FUNCTION_BLOCK FB_ECS_Linear_AO
VAR_INPUT PERSISTENT
	bEnable									: BOOL;											//{#lynus.ag#()} //Enable the Fuctionblock and his logic
	bPowerDataInvers						: BOOL;											//With True its possible to invert all received power data from the electric meter
	bNoLinear								: BOOL;											//Output Power from the device is not linear. Use the Values from the Table Of Interpolation Points.
	byElectricFuseLine						: BYTE; 										//Electric Fuse Line on wich the ECS is connected => 1 2 3 (If 0 then this charging station is not connected to a Electric Fuse Line)
	diNrOfEMS_IN							: DINT;											//Number of EMS what control this Device.
	diNrOfEM_IN_CS							: DINT;											//Number of the electric meter for incoming power data. (Power Data for this Device)
	stSetupECS								: ST_Setup_ECS;									//{#lynus.ag#()} //Setup charging station
	arrTableOfInterpolationPoints			: ARRAY[1..10] OF REAL;							//Table Of Interpolation Points. Corresponds to the different power values in the non-linear curve of the device. The last value must correspond to the maximum power.
END_VAR
VAR_INPUT
	bCarConnectedExt						: BOOL;											//Car connected signal from external function			
	bErrorExt								: BOOL;											//Error Signal from external Function
	bWarningExt								: BOOL;											//Warning Signal from external Function 						
END_VAR
VAR_OUTPUT
	stDataECS								: ST_ECS_Output;								//{#lynus.ag#()} //Electric charging station output data
	diNrOfECS_OUT							: DINT;											//Active Number from the Electric charging Function for using on other functions
	rTargetPowerForExtFunc					: REAL;											//Target Power from 0% to +100% to use on a external Function
	rTargetChargCurrentForExtFunc			: REAL;											//Target charge Current to use on a external Function
END_VAR
VAR
	{attribute 'hide'}
	fbCS									: FB_ElectricChargingStation;					//Function block for electric charging station
	{attribute 'hide'}
	fbNumberDevice							: FB_NumberOfDevice;							//Function block to calcualte the number of the Device
	{attribute 'hide'}
	fbInterpolation							: FB_Lin_Interpolation;							//Function for interpolation
	fbDIExternalLock						: FB_XL1XXX_DI;									//Digital Input from external loock signal
	fbAOCS									: FB_XL4XXX_AO;									//Analog Output to swtich on and off the charging station
	{attribute 'hide'}
	timDissableFunctions					: TON;											//Timer to dissable the Function after Lynus_Standards.Constants_General.tTimeDissableLynusFunctions Days without connection to the Lynus Cloud
	{attribute 'hide'}
	timResetConnectionOnGVL					: TON;											//Timer to try reset the connection Flag on the GVL. (When somebody delete the Connection Function and make only a onlinechange)
	{attribute 'hide'}
	arrPD									: ARRAY[1..25] OF FB_PersistentData_Number;		//Function to save persistent data 
	{attribute 'hide'}
	byWaitInStep							: BYTE;											//Wait in Step before start to clean data on PLC
	{attribute 'hide'}
	iStateGVLData							: INT;											//State machine to handle the data on the GVL
	{attribute 'hide'}
	diNumberOfActiveBatterys				: DINT;											//Number of active batterys
	{attribute 'hide'}
	diNumberOfBatteryInverterInEPO			: DINT;											//Number of battery inverters that work in Emergency Power operation 
	{attribute 'hide'}
	diCounterForGVL							: DINT;											//Counter to clean old data on GVL
	{attribute 'hide'}
	diLPForGVL								: DINT;											//Loop to clean old data on GVL
	{attribute 'hide'}
	dwSumSOC								: DWORD;										//Sum of the SOC from all batterys	
	{attribute 'hide'}
	liLPBatteryData							: LINT;											//Loop to check some data from batterys
	{attribute 'hide'}
	liLPInEPO								: LINT;											//Loop to check if 1 or more battery inverters build a island grid
END_VAR
VAR PERSISTENT
	{attribute 'conditionalshow'}
	diNrOfEMS_IN_CP							: DINT;											//Number of EMS what control this Device to compare with the original
END_VAR

//Creator : Kai Ebensperger
//Company : Lynus AG
//Date : 19.05.2021
//Version : 1.0.0.0

//With this function block its possible to switch on and off a charging station
//Its also possible to control the target power with the analog output signal
//With the Nr from the Electric Meter its possible to send the data fromt the electric meter directly to the CS function to display it

//NOTE for diNr.....Designation => 
//_IN = Here Data come in from other Functions or go out to other functions about the GVL
//_OUT = Here Data go out to other functions about the GVL

(*------------------------------------------------------------Limits----------------------------------------------------------------------------------*)

diNrOfEMS_IN := LIMIT(0,diNrOfEMS_IN,Constants_Energy.diMaxNumberOfEMS);
	diNrOfEM_IN_CS := LIMIT(0,diNrOfEM_IN_CS,Constants_Energy.diMaxNumberOfElectricMeters);	
		byElectricFuseLine := LIMIT(0,byElectricFuseLine,30);	
			
(*------------------------------------------------------------------Power Data----------------------------------------------------------------------------*)

//Energy Session Input data
fbCS.bCalculateEnergySession := FALSE;
fbCS.arrSocketPowerECS[1] := 0;
fbCS.arrSocketPowerECS[2] := 0;
fbCS.arrSocketPowerECS[3] := 0;
fbCS.arrSocketPowerECS[4] := 0;
fbCS.arrSocketEnergySession[1] := 0;
fbCS.arrSocketEnergySession[2] := 0;
fbCS.arrSocketEnergySession[3] := 0;
fbCS.arrSocketEnergySession[4] := 0;

IF NOT bPowerDataInvers THEN
	fbCS.lrCounterEnergyT1_Consumption := Lynus_Standards.GVL_Energy.stDataElectricMeters[diNrOfEM_IN_CS].lrCounterEnergyT1_Production * 1000;
	fbCS.lrCounterEnergyT2_Consumption := Lynus_Standards.GVL_Energy.stDataElectricMeters[diNrOfEM_IN_CS].lrCounterEnergyT2_Production * 1000;
	fbCS.lrCounterEnergyT1_Production := Lynus_Standards.GVL_Energy.stDataElectricMeters[diNrOfEM_IN_CS].lrCounterEnergyT1_Consumption * 1000;
	fbCS.lrCounterEnergyT2_Production := Lynus_Standards.GVL_Energy.stDataElectricMeters[diNrOfEM_IN_CS].lrCounterEnergyT1_Consumption * 1000;
	fbCS.lrTotalCounterEnergy_Consumption := Lynus_Standards.GVL_Energy.stDataElectricMeters[diNrOfEM_IN_CS].lrTotalCounterEnergy_Production * 1000;
	fbCS.lrTotalCounterEnergy_Production := Lynus_Standards.GVL_Energy.stDataElectricMeters[diNrOfEM_IN_CS].lrTotalCounterEnergy_Consumption * 1000;
		fbCS.lrTotalPowerECS := (Lynus_Standards.GVL_Energy.stDataElectricMeters[diNrOfEM_IN_CS].lrPower * 1000) * - 1;
ELSE
	fbCS.lrCounterEnergyT1_Consumption := Lynus_Standards.GVL_Energy.stDataElectricMeters[diNrOfEM_IN_CS].lrCounterEnergyT1_Consumption * 1000;
	fbCS.lrCounterEnergyT2_Consumption := Lynus_Standards.GVL_Energy.stDataElectricMeters[diNrOfEM_IN_CS].lrCounterEnergyT2_Consumption * 1000;
	fbCS.lrCounterEnergyT1_Production := Lynus_Standards.GVL_Energy.stDataElectricMeters[diNrOfEM_IN_CS].lrCounterEnergyT1_Production * 1000;
	fbCS.lrCounterEnergyT2_Production := Lynus_Standards.GVL_Energy.stDataElectricMeters[diNrOfEM_IN_CS].lrCounterEnergyT2_Production * 1000;
	fbCS.lrTotalCounterEnergy_Consumption := Lynus_Standards.GVL_Energy.stDataElectricMeters[diNrOfEM_IN_CS].lrTotalCounterEnergy_Consumption * 1000;
	fbCS.lrTotalCounterEnergy_Production := Lynus_Standards.GVL_Energy.stDataElectricMeters[diNrOfEM_IN_CS].lrTotalCounterEnergy_Production * 1000;
		fbCS.lrTotalPowerECS := Lynus_Standards.GVL_Energy.stDataElectricMeters[diNrOfEM_IN_CS].lrPower * 1000;
END_IF

(*-------------------------------------------------------------Calcualte the number of ECS---------------------------------------------------------------*)

fbNumberDevice(
	diActualNumberOfDevices:= Lynus_Standards.GVL_Energy.stNumberOfDevices.diNumberOfECS, 
	diMaxNumberOfDevices:= Constants_Energy.diMaxNumberOfElectricChargingStations, 
	udiCounterOnlineChange:= TwinCAT_SystemInfoVarList._AppInfo.OnlineChangeCnt, 
	bNumberIsCalculatet=> , 
	bFPNumberIsCalculatet=> , 
	bOnlineChange=> , 
	diNumberForThisDevice=> diNrOfECS_OUT, 
	diNumberOfTotalDevices=> );

//Write new Numer on GVL
IF fbNumberDevice.bFPNumberIsCalculatet THEN
	Lynus_Standards.GVL_Energy.stNumberOfDevices.diNumberOfECS := fbNumberDevice.diNumberOfTotalDevices;	
END_IF 

//Delete old Number on GVL
IF fbNumberDevice.bOnlineChange THEN 
	Lynus_Standards.GVL_Energy.stNumberOfDevices.diNumberOfECS := diNrOfECS_OUT;	
		iStateGVLData := 1; 
END_IF

(*-------------------------------------------------------------Service from Backend is ready and check the connection to backend for dissabel/enable Function---------------------------------------------------------------*)

//Try to reset the variable for connection on the GVL. When all is normal then the Lynus Mqtt connection function set this variable to true in the next cycle
//When we have no connection to the backend then after Lynus_Standards.Constants_General.tTimeDissableLynusFunctions days the Function is dissabled with all of his functionalities
timResetConnectionOnGVL(IN:= NOT timResetConnectionOnGVL.Q, PT:= T#1H, Q=> , ET=> );
	IF timResetConnectionOnGVL.Q THEN Lynus_Standards.GVL_Communicator.bStateConnectionToEnableFunctions := FALSE; END_IF
		IF NOT Lynus_Standards.GVL_Communicator.bStateConnectionToEnableFunctions THEN timDissableFunctions.IN := TRUE; ELSE timDissableFunctions.IN := FALSE; END_IF  
			timDissableFunctions(IN:= , PT:= Lynus_Standards.Constants_General.tTimeDissableLynusFunctions, Q=> , ET=> );	

(*------------------------------------------------------------------Error and Warning----------------------------------------------------------------------------*)	

IF timDissableFunctions.Q OR bWarningExt THEN fbCS.bWarning := TRUE; ELSE fbCS.bWarning := FALSE; END_IF   
	IF Lynus_Standards.GVL_Energy.stNumberOfDevices.diNumberOfECS > Constants_Energy.diMaxNumberOfElectricChargingStations OR bErrorExt THEN 
		fbCS.bError := TRUE;
	ELSE 
		fbCS.bError := FALSE;
	END_IF

IF timDissableFunctions.Q THEN fbCS.iWarningCode := 0;
ELSIF bWarningExt THEN fbCS.iWarningCode := 1;
END_IF

IF Lynus_Standards.GVL_Energy.stNumberOfDevices.diNumberOfECS > Constants_Energy.diMaxNumberOfElectricChargingStations THEN fbCS.iErrorCode := 1;
ELSIF bErrorExt THEN fbCS.iErrorCode := 0;
END_IF        	
	
(*------------------------------------------------------------------Logic----------------------------------------------------------------------------*)

//Calcualte the total SOC if we have more then 1 battery in our system
diNumberOfActiveBatterys := 0;
	dwSumSOC := 0;
		FOR liLPBatteryData := 1 TO Constants_Energy.diMaxNumberOfBatterys BY 1 DO
			IF Lynus_Standards.GVL_Energy.stDataOfBatterys[diNrOfEMS_IN,liLPBatteryData].bEnabled THEN diNumberOfActiveBatterys := diNumberOfActiveBatterys + 1; END_IF
				dwSumSOC := dwSumSOC + Lynus_Standards.GVL_Energy.stDataOfBatterys[diNrOfEMS_IN,liLPBatteryData].dwSOC;
		END_FOR
	
IF diNumberOfActiveBatterys > 0 THEN
	fbCS.dwBatterySOC := DINT_TO_DWORD(DWORD_TO_DINT(dwSumSOC) / diNumberOfActiveBatterys);
ELSE
	fbCS.dwBatterySOC := 100;	//When we have no battery in the ems system
END_IF

//Check if one or more Batterysystems or batteryinverter make island mode
diNumberOfBatteryInverterInEPO := 0;
	FOR liLPInEPO := 1 TO Constants_Energy.diMaxNumberOfBatteryInverters BY 1 DO
		IF Lynus_Standards.GVL_Energy.stDataOfBatteryInverters[diNrOfEMS_IN,liLPInEPO].bWorkOnIslandMode THEN fbCS.bEPOIsActive := TRUE; diNumberOfBatteryInverterInEPO := diNumberOfBatteryInverterInEPO + 1; END_IF
	END_FOR 
		IF diNumberOfBatteryInverterInEPO <= 0 THEN fbCS.bEPOIsActive := FALSE; END_IF

//Digital input for external lock signal
fbDIExternalLock(bInvers:= FALSE, bSignal=> );

//Car SOC, charging Time and Mode 3
fbCS.arrSOCCar[1] := 0;
fbCS.arrSOCCar[2] := 0;
fbCS.arrSOCCar[3] := 0;
fbCS.arrSOCCar[4] := 0;
	fbCS.arrSocketChargingTimeInput[1] := 0;
	fbCS.arrSocketChargingTimeInput[2] := 0;
	fbCS.arrSocketChargingTimeInput[3] := 0;
	fbCS.arrSocketChargingTimeInput[4] := 0;
		fbCS.arrSocketMode3StateECS[1] := '';
		fbCS.arrSocketMode3StateECS[2] := '';
		fbCS.arrSocketMode3StateECS[3] := '';
		fbCS.arrSocketMode3StateECS[4] := '';
	
//Functionblock ECS
fbCS(
	bEnable:= bEnable AND NOT timDissableFunctions.Q, 
	bError:= , 
	bEPOIsActive:= , 
	bExternalLock:= fbDIExternalLock.bSignal, 
	bCarConnected:= bCarConnectedExt, 
	bWriteWithDelay:= TRUE, 
	bCalculateEnergySession:= ,
	iErrorCode:= , 
	iWarningCode:= , 
	arrSocketChargingTimeInput:= , 
	arrSOCCar:= , 
	dwBatterySOC:= , 
	lrTotalCounterEnergy_Consumption:= , 
	lrTotalCounterEnergy_Production:= , 
	lrCounterEnergyT1_Consumption:= , 
	lrCounterEnergyT2_Consumption:= , 
	lrCounterEnergyT1_Production:= , 
	lrCounterEnergyT2_Production:= , 
	lrTotalPowerECS:= , 
	arrSocketEnergySession:= ,
	rTargetPower:= Lynus_Standards.GVL_Energy.stDataElectricChargingStations[diNrOfEMS_IN,diNrOfECS_OUT].rTargetPowerEMS, 
	rSupplyVoltage:= 692, 
	rMinCurrent:= 0, 
	tTimDelayOutput:= T#5S, 
	tDelayError:= T#5S,
	arrSocketMode3StateECS:= ,
	arrSocketPowerECS:= ,
	stSetupECS:= stSetupECS, 
	stDataECSOut=> , 
	stDataECSOutDelay=> stDataECS);	
	
(*-------------------------------------------------------------------------Output----------------------------------------------------------------------*)

IF bNoLinear THEN 
	fbInterpolation.rXInputValue := (stSetupECS.rMaxPower * fbCS.stDataECSOut.rTargetPower) / 100; 
		fbInterpolation.arrYIntermediateValues[1] := 10;
			fbInterpolation.arrYIntermediateValues[2] := 20;
				fbInterpolation.arrYIntermediateValues[3] := 30;
					fbInterpolation.arrYIntermediateValues[4] := 40;
						fbInterpolation.arrYIntermediateValues[5] := 50;
	fbInterpolation.arrYIntermediateValues[6] := 60;
		fbInterpolation.arrYIntermediateValues[7] := 70;
			fbInterpolation.arrYIntermediateValues[8] := 80;
				fbInterpolation.arrYIntermediateValues[9] := 90;
					fbInterpolation.arrYIntermediateValues[10] := 100;
	fbInterpolation(rXInputValue:=, arrXIntermediateValues:= arrTableOfInterpolationPoints, arrYIntermediateValues:=, rYOutputValue=> );
END_IF

IF bNoLinear THEN 
	fbAOCS.rSignal := fbInterpolation.rYOutputValue;
	//Target Power, to use this on a external Function
	rTargetPowerForExtFunc := fbInterpolation.rYOutputValue;
	rTargetChargCurrentForExtFunc := (fbCS.stDataECSOut.rTargetChargeCurrent * rTargetPowerForExtFunc) / 100; 
ELSE
	fbAOCS.rSignal := fbCS.stDataECSOut.rTargetPower;
	//Target Power, to use this on a external Function
	rTargetPowerForExtFunc := fbCS.stDataECSOut.rTargetPower;
	rTargetChargCurrentForExtFunc := fbCS.stDataECSOut.rTargetChargeCurrent;
END_IF

fbAOCS(
	rYMinTerminalValue:= 0, 
	rXMinInputSignal:= 0, 
	rYMaxTerminalValue:= 32767, 
	rXMaxInputSignal:= 100, 
	rSignal:= , 
	usiState=> );
							
(*-----------------------------------------------------------Handle data to Global structure for electric charging stations-----------------------------------------------------------------*)

//Delte al old Data on GVL after a online change or change on the variable diNrOfEMS_IDOD
IF diNrOfEMS_IN <> diNrOfEMS_IN_CP AND iStateGVLData = 0 THEN iStateGVLData := 10; END_IF 

CASE iStateGVLData OF
	
	0://Init Step
		byWaitInStep := 0;
			diCounterForGVL := 1;
	
	1://Wait for 4 Steps before clean al Data on GVL
		byWaitInStep := byWaitInStep + 1;
			IF byWaitInStep >= 4 AND fbNumberDevice.bNumberIsCalculatet THEN iStateGVLData := 2; END_IF
				//To much Devices, back to the Init step
				IF byWaitInStep >= 4 AND NOT fbNumberDevice.bNumberIsCalculatet THEN iStateGVLData := 0; END_IF	
			
	2://Clear all Data in GVL
		FOR diLPForGVL := 1 TO Constants_Energy.diMaxNumberOfEMS BY 1 DO 
			Lynus_Standards.GVL_Energy.stDataElectricChargingStations[diLPForGVL,diCounterForGVL].bEnabled := FALSE;
				Lynus_Standards.GVL_Energy.stDataElectricChargingStations[diLPForGVL,diCounterForGVL].bIsControllable := FALSE;
					Lynus_Standards.GVL_Energy.stDataElectricChargingStations[diLPForGVL,diCounterForGVL].byErrorWarning := 0;
						Lynus_Standards.GVL_Energy.stDataElectricChargingStations[diLPForGVL,diCounterForGVL].byPriority := 0;
							Lynus_Standards.GVL_Energy.stDataElectricChargingStations[diLPForGVL,diCounterForGVL].lrPower := 0;
								Lynus_Standards.GVL_Energy.stDataElectricChargingStations[diLPForGVL,diCounterForGVL].lrPowerConsumption := 0;
									Lynus_Standards.GVL_Energy.stDataElectricChargingStations[diLPForGVL,diCounterForGVL].lrPowerProduction := 0;
										Lynus_Standards.GVL_Energy.stDataElectricChargingStations[diLPForGVL,diCounterForGVL].rMaxPower := 0;
											Lynus_Standards.GVL_Energy.stDataElectricChargingStations[diLPForGVL,diCounterForGVL].byElectricFuseLine := 0;
												//Set also the target value from ems back here to 0 and not in EMS function because EMS is in Standy when we have a online change (Problem when we delete a ems function and make a online change)
												Lynus_Standards.GVL_Energy.stDataElectricChargingStations[diLPForGVL,diCounterForGVL].rTargetPowerEMS := 0;	
		END_FOR
			diCounterForGVL := diCounterForGVL + 1;
				diCounterForGVL := LIMIT(0,diCounterForGVL,Constants_Energy.diMaxNumberOfElectricChargingStations);
					//Back to the init step
					IF diCounterForGVL >= Constants_Energy.diMaxNumberOfElectricChargingStations THEN iStateGVLData := 0; END_IF

	10://Clear old Data on GVL 		
		Lynus_Standards.GVL_Energy.stDataElectricChargingStations[diNrOfEMS_IN_CP,diNrOfECS_OUT].bEnabled := FALSE;
			Lynus_Standards.GVL_Energy.stDataElectricChargingStations[diNrOfEMS_IN_CP,diNrOfECS_OUT].bIsControllable := FALSE;
				Lynus_Standards.GVL_Energy.stDataElectricChargingStations[diNrOfEMS_IN_CP,diNrOfECS_OUT].byErrorWarning := 0;
					Lynus_Standards.GVL_Energy.stDataElectricChargingStations[diNrOfEMS_IN_CP,diNrOfECS_OUT].byPriority := 0;
						Lynus_Standards.GVL_Energy.stDataElectricChargingStations[diNrOfEMS_IN_CP,diNrOfECS_OUT].lrPower := 0;
							Lynus_Standards.GVL_Energy.stDataElectricChargingStations[diNrOfEMS_IN_CP,diNrOfECS_OUT].lrPowerConsumption := 0;
								Lynus_Standards.GVL_Energy.stDataElectricChargingStations[diNrOfEMS_IN_CP,diNrOfECS_OUT].lrPowerProduction := 0;
									Lynus_Standards.GVL_Energy.stDataElectricChargingStations[diNrOfEMS_IN_CP,diNrOfECS_OUT].rMaxPower := 0;
										Lynus_Standards.GVL_Energy.stDataElectricChargingStations[diNrOfEMS_IN_CP,diNrOfECS_OUT].byElectricFuseLine := 0;
									
		diNrOfEMS_IN_CP := diNrOfEMS_IN;
			//Back to the init step
			iStateGVLData := 0;

END_CASE 	 

IF diNrOfECS_OUT > 0 AND fbNumberDevice.bNumberIsCalculatet AND diNrOfEMS_IN > 0 THEN
	Lynus_Standards.GVL_Energy.stDataElectricChargingStations[diNrOfEMS_IN,diNrOfECS_OUT].bEnabled := fbCS.stDataECSOut.bEnabled;
		Lynus_Standards.GVL_Energy.stDataElectricChargingStations[diNrOfEMS_IN,diNrOfECS_OUT].bIsControllable := TRUE;
			Lynus_Standards.GVL_Energy.stDataElectricChargingStations[diNrOfEMS_IN,diNrOfECS_OUT].byErrorWarning := fbCS.stDataECSOut.byErrorWarning;
				Lynus_Standards.GVL_Energy.stDataElectricChargingStations[diNrOfEMS_IN,diNrOfECS_OUT].byPriority := fbCS.stDataECSOut.byPriority;
					Lynus_Standards.GVL_Energy.stDataElectricChargingStations[diNrOfEMS_IN,diNrOfECS_OUT].lrPower := fbCS.stDataECSOut.lrTotalPower;
						Lynus_Standards.GVL_Energy.stDataElectricChargingStations[diNrOfEMS_IN,diNrOfECS_OUT].lrPowerConsumption := fbCS.stDataECSOut.lrTotalPowerConsumption;
							Lynus_Standards.GVL_Energy.stDataElectricChargingStations[diNrOfEMS_IN,diNrOfECS_OUT].lrPowerProduction := fbCS.stDataECSOut.lrTotalPowerProduction;
								Lynus_Standards.GVL_Energy.stDataElectricChargingStations[diNrOfEMS_IN,diNrOfECS_OUT].rMaxPower := fbCS.stDataECSOut.rMaxPower;	
									Lynus_Standards.GVL_Energy.stDataElectricChargingStations[diNrOfEMS_IN,diNrOfECS_OUT].byElectricFuseLine := byElectricFuseLine;	
END_IF 
		
(*----------------------------------------------------------Save persistent data----------------------------------------------------------------*)

arrPD[1](lrValue:= BOOL_TO_LREAL(bEnable), bEventBasedActive=> );
arrPD[2](lrValue:= BOOL_TO_LREAL(bPowerDataInvers), bEventBasedActive=> );
arrPD[3](lrValue:= DINT_TO_LREAL(diNrOfEMS_IN), bEventBasedActive=> );
arrPD[4](lrValue:= DINT_TO_LREAL(diNrOfEM_IN_CS), bEventBasedActive=> );
arrPD[5](lrValue:= BOOL_TO_LREAL(stSetupECS.bManualyOn), bEventBasedActive=> );
arrPD[6](lrValue:= BOOL_TO_LREAL(stSetupECS.bOnEmergPowerOff), bEventBasedActive=> );
arrPD[7](lrValue:= BYTE_TO_LREAL(stSetupECS.byCSMinPower), bEventBasedActive=> );
arrPD[8](lrValue:= BYTE_TO_LREAL(stSetupECS.byDisableSOC), bEventBasedActive=> );
arrPD[9](lrValue:= BYTE_TO_LREAL(stSetupECS.byEnableSOC), bEventBasedActive=> );
arrPD[10](lrValue:= BYTE_TO_LREAL(stSetupECS.byManualyTargetPower), bEventBasedActive=> );
arrPD[11](lrValue:= BYTE_TO_LREAL(stSetupECS.byPriority), bEventBasedActive=> );
arrPD[12](lrValue:= REAL_TO_LREAL(stSetupECS.rMaxPower), bEventBasedActive=> );
arrPD[13](lrValue:= DINT_TO_LREAL(diNrOfEMS_IN_CP), bEventBasedActive=> );
arrPD[14](lrValue:= BOOL_TO_LREAL(bNoLinear), bEventBasedActive=> );
arrPD[15](lrValue:= REAL_TO_LREAL(arrTableOfInterpolationPoints[1]), bEventBasedActive=> );
arrPD[16](lrValue:= REAL_TO_LREAL(arrTableOfInterpolationPoints[2]), bEventBasedActive=> );
arrPD[17](lrValue:= REAL_TO_LREAL(arrTableOfInterpolationPoints[3]), bEventBasedActive=> );
arrPD[18](lrValue:= REAL_TO_LREAL(arrTableOfInterpolationPoints[4]), bEventBasedActive=> );
arrPD[19](lrValue:= REAL_TO_LREAL(arrTableOfInterpolationPoints[5]), bEventBasedActive=> );
arrPD[20](lrValue:= REAL_TO_LREAL(arrTableOfInterpolationPoints[6]), bEventBasedActive=> );
arrPD[21](lrValue:= REAL_TO_LREAL(arrTableOfInterpolationPoints[7]), bEventBasedActive=> );
arrPD[22](lrValue:= REAL_TO_LREAL(arrTableOfInterpolationPoints[8]), bEventBasedActive=> );
arrPD[23](lrValue:= REAL_TO_LREAL(arrTableOfInterpolationPoints[9]), bEventBasedActive=> );
arrPD[24](lrValue:= REAL_TO_LREAL(arrTableOfInterpolationPoints[10]), bEventBasedActive=> );
arrPD[25](lrValue:= BYTE_TO_LREAL(byElectricFuseLine), bEventBasedActive=> );

END_FUNCTION_BLOCK

(* stored: Version 1.1.0.1, ProductVersion 3.1.4024.9
   POU FB_ECS_Linear_AO: Id {4879927e-0a5c-45f1-8b4c-68c3bf0795b3}, SpecialFunc None *)
